TYPE ST_3005_GoToDestination EXTENDS ST_SupervisorHeader :
	STRUCT
		DestinationID : UDINT;
	END_STRUCT
END_TYPE

(* stored: Version 1.1.0.1
   DUT ST_3005_GoToDestination: Id {59e26304-7ab2-48dc-acd6-0a8e75d3cbc7} *)
